PROGRAM prgHouse
VAR
	lrPowerHouse		: LREAL;						//{#lynus.ag#()}
	bEnableHouse		: BOOL;					//{#lynus.ag#()}
	bHouseEnabled		: BOOL;;					//{#lynus.ag#()}

END_VAR

lrPowerHouse			:=	prg_ADS.struct_received.lrPowerHouse			;
bEnableHouse			:=	prg_ADS.struct_received.bEnableHouse			;
bHouseEnabled			:=	prg_ADS.struct_received.bHouseEnabled			;

END_PROGRAM

(* stored: Version 1.1.0.1, ProductVersion 3.1.4024.12
   POU prgHouse: Id {32a50f47-0b6d-4649-94c0-50dfea60d5bd}, SpecialFunc None *)
